TYPE ST_Machine_HMI :
	STRUCT
		Cmd : ST_Machine_Cmd;
		Cfg : ST_Machine_Cfg;
		Sts : ST_Machine_Sts;
	END_STRUCT
END_TYPE

(* stored: Version 1.1.0.1
   DUT ST_Machine_HMI: Id {d8e87d17-7eba-4b6b-b7ba-5a1315b120d0} *)
